Xinje XDPPro project, PLC1: XD5-48T6 (software 3.5.3 2018-11-19)

PROGRAM Ladder

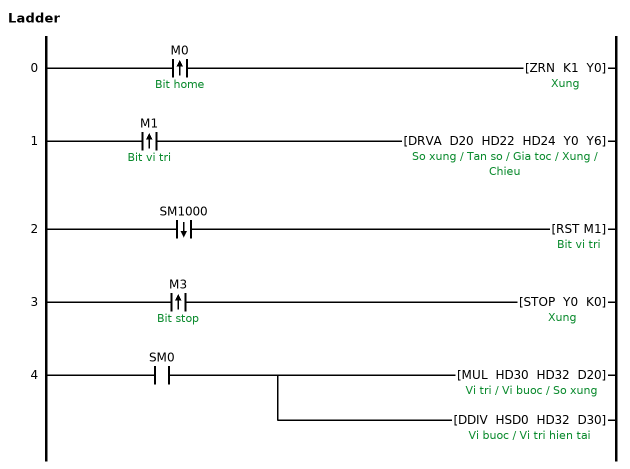
LDP    M0	; Bit home
ZRN    K1 Y0	; Xung
LDP    M1	; Bit vi tri
DRVA   D20 HD22 HD24 Y0 Y6	; So xung / Tan so / Gia toc / Xung / Chieu
LDF    SM1000
RST    M1	; Bit vi tri
LDP    M3	; Bit stop
STOP   Y0 K0	; Xung
LD     SM0
MUL    HD30 HD32 D20	; Vi tri / Vi buoc / So xung
DDIV   HSD0 HD32 D30	; Vi buoc / Vi tri hien tai